PROGRAM TSCS_Bridge_Test
VAR
	// Bridge Test - Fast counter
	RS_0: RS;	
	CountUp_Act : BOOL;
	Counter : REAL;
	
	Counter_RB_Diff : REAL;
	
	Counter_LL : REAL := -5000.0;
	Counter_UL : REAL := 5000.0;
END_VAR
VAR // added by the converter: edge detectors and wires of the graphical bodies
    _rt1, _rt2 : R_TRIG;
END_VAR

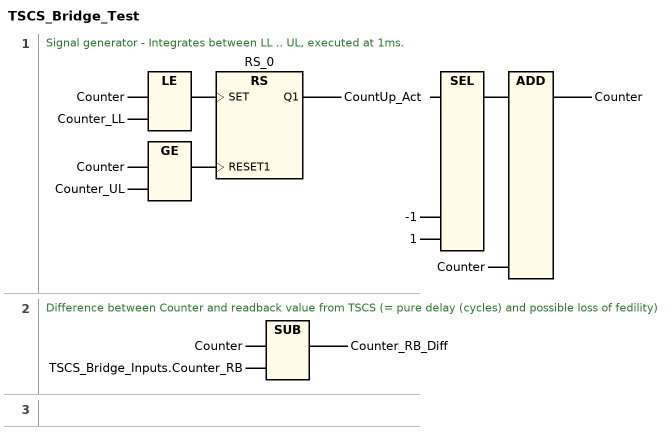
// NETWORK 1
// Signal generator - Integrates between LL .. UL, executed at 1ms.
_rt1(CLK := Counter <= Counter_LL);
_rt2(CLK := Counter >= Counter_UL);
RS_0(SET := _rt1.Q, RESET1 := _rt2.Q); // RS
CountUp_Act := RS_0.Q1;
Counter := SEL(RS_0.Q1, -1, 1) + Counter;

// NETWORK 2
// Difference between Counter and readback value from TSCS (= pure delay (cycles) and possible loss of fedility)
Counter_RB_Diff := Counter - TSCS_Bridge_Inputs.Counter_RB;

// NETWORK 3

END_PROGRAM

(* stored: Version 1.1.0.1, ProductVersion 3.1.4024.6
   POU TSCS_Bridge_Test: Id {c2404466-5f35-444f-8eba-adf42f60161e}, SpecialFunc None *)
